{attribute 'qualified_only'}
VAR_GLOBAL
	fPayloadHeightIni: LREAL := 0.0;
END_VAR

(* stored: Version 1.1.0.1, ProductVersion 3.1.4024.12
   GVL GVL_WinchHeightControl: Id {eaddd7bf-d6bd-481d-8985-3b578109bf07} *)
